RoboDK station: UR3e only.rdk

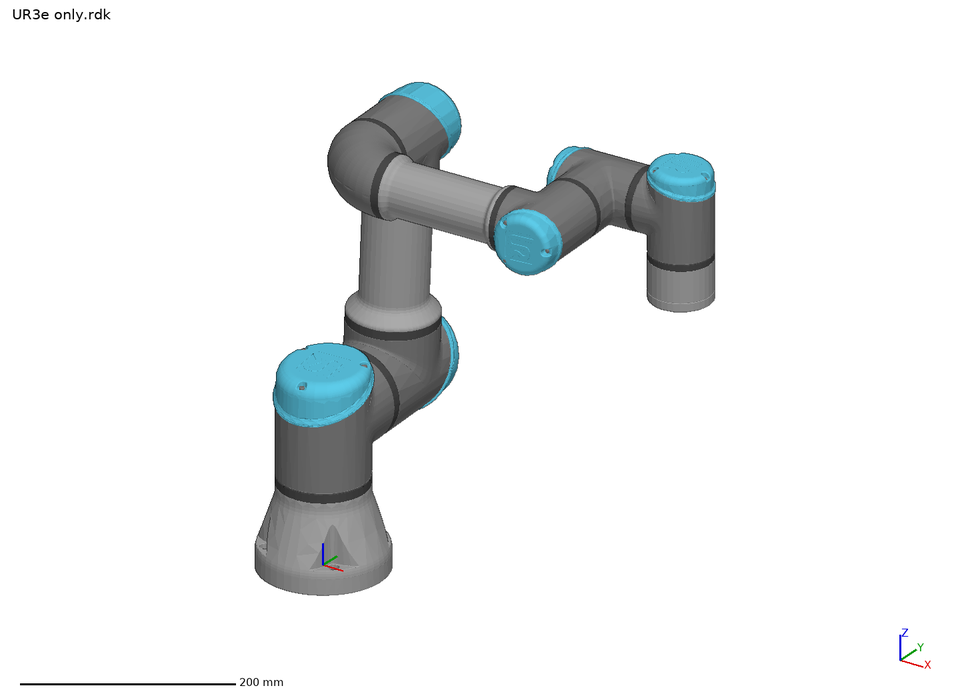
[picture v0: the station drawn from its stored meshes, robots at their saved joint values, targets as dots, program paths as lines]
Station UR3e only (saved by RoboDK 5.9.5). Poses are relative to the parent item; angles as X-Y-Z fixed-axis rotations.
Station parameters (name, value as stored): OPC-UA, opc.tcp://localhost:4840
  - frame UR3e Base at (0, 0, 0) mm
    - robot UR3e: 6 axes, payload 3 kg, reach 500 mm, repeatability 0.03 mm, weight 11 kg
        modified DH rows (alpha deg, a mm, theta deg, d mm): 0, 0, 0, 151.9; 90, 0, 180, 0; 0, 243.55, 0, 0; 0, 213.2, 0, 131.05; -90, 0, 0, 85.35; 90, 0, 180, 92.1
        joint limits [-360, -360, -360, -360, -360, -360] to [360, 360, 360, 360, 360, 360]; home [0, -90, -90, 0, 90, 0]; saved at [183.566, -87.595, 88.437, -90.843, -90, -86.434]
  - Python program Prog1 (listed below)
  - Python program SampleOfflineProgramming (listed below)

--- Python program Prog1 ---
# Type help("robodk.robolink") or help("robodk.robomath") for more information
# Press F5 to run the script
# Documentation: https://robodk.com/doc/en/RoboDK-API.html
# Reference:     https://robodk.com/doc/en/PythonAPI/robodk.html
# Note: It is not required to keep a copy of this file, your Python script is saved with your RDK project

from robodk.robolink import *
from robodk.robomath import *

RDK = Robolink()

# Roboter holen
robot = RDK.Item('UR3e', ITEM_TYPE_ROBOT)

if not robot.Valid():
    raise Exception("Roboter 'UR3e' nicht gefunden")

# Geschwindigkeit
robot.setSpeed(100)

# Zwei Posen definieren
pose_1 = transl(300, -150, 300) * rotx(pi)
pose_2 = transl(300,  150, 300) * rotx(pi)

# Startposition
robot.MoveJ([0, -90, 90, -90, -90, 0])

# Abwechselnd zwei Posen anfahren
for i in range(5):
    robot.MoveJ(pose_1)
    pause(1)

    robot.MoveJ(pose_2)
    pause(1)

--- Python program SampleOfflineProgramming ---
# This macro shows an example to draw a polygon of radius R and n_sides vertices using the RoboDK API for Python
# More information about the RoboDK API here:
# https://robodk.com/doc/en/RoboDK-API.html
from robodk.robolink import *  # API to communicate with RoboDK
from robodk.robomath import *  # basic matrix operations

# Any interaction with RoboDK must be done through RDK:
RDK = Robolink()

# Select a robot (popup is displayed if more than one robot is available)
robot = RDK.ItemUserPick('Select a robot', ITEM_TYPE_ROBOT)
if not robot.Valid():
    raise Exception('No robot selected or available')

# get the current position of the TCP with respect to the reference frame:
# (4x4 matrix representing position and orientation)
target_ref = robot.Pose()
pos_ref = target_ref.Pos()
print("Drawing a polygon around the target: ")
print(Pose_2_TxyzRxyz(target_ref))

# move the robot to the first point:
robot.MoveJ(target_ref)

# It is important to provide the reference frame and the tool frames when generating programs offline
robot.setPoseFrame(robot.PoseFrame())
robot.setPoseTool(robot.PoseTool())
robot.setRounding(10)  # Set the rounding parameter (Also known as: CNT, APO/C_DIS, ZoneData, Blending radius, cornering, ...)
robot.setSpeed(200)  # Set linear speed in mm/s

# Set the number of sides of the polygon:
n_sides = 6
R = 100

# make a hexagon around reference target:
for i in range(n_sides + 1):
    ang = i * 2 * pi / n_sides  #angle: 0, 60, 120, ...

    #-----------------------------
    # Movement relative to the reference frame
    # Create a copy of the target
    target_i = Mat(target_ref)
    pos_i = target_i.Pos()
    pos_i[0] = pos_i[0] + R * cos(ang)
    pos_i[1] = pos_i[1] + R * sin(ang)
    target_i.setPos(pos_i)
    print("Moving to target %i: angle %.1f" % (i, ang * 180 / pi))
    print(str(Pose_2_TxyzRxyz(target_i)))
    robot.MoveL(target_i)

    #-----------------------------
    # Post multiply: relative to the tool
    #target_i = target_ref * rotz(ang) * transl(R,0,0) * rotz(-ang)
    #robot.MoveL(target_i)

# move back to the center, then home:
robot.MoveL(target_ref)

print('Done')
